INTERFACE I_Base EXTENDS __SYSTEM.IQUERYINTERFACE

END_INTERFACE

(* stored: Version 1.1.0.1
   Itf I_Base: Id {8863f417-84d9-475b-8ed5-cfaf8d0a02ca} *)
